PROGRAM P2_05_Process_Ctrl
VAR
	bWaitAferBatchClose			:BOOL;
	tonWaitAfterBatchClose		:TON;
END_VAR
VAR // added by the converter: edge detectors and wires of the graphical bodies
    _w1, _w2, _w3, _w4, _w5, _w6, _w7, _w8, _w9 : BOOL;
    _rt1, _rt2 : R_TRIG;
END_VAR

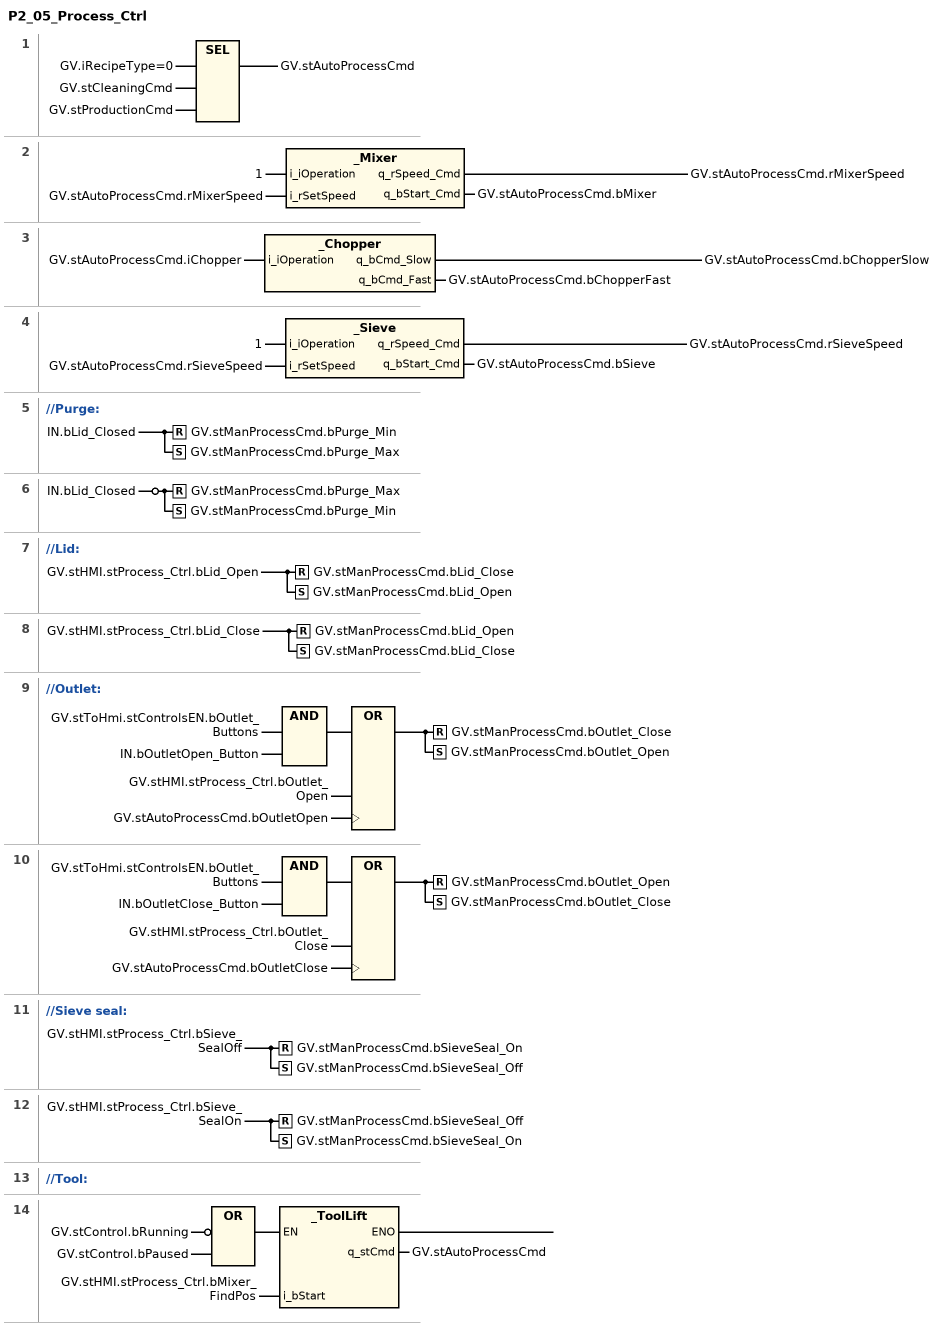
// NETWORK 1
GV.stAutoProcessCmd := SEL(GV.iRecipeType=0, GV.stCleaningCmd, GV.stProductionCmd);

// NETWORK 2
_Mixer(i_iOperation := 1, i_rSetSpeed := GV.stAutoProcessCmd.rMixerSpeed, q_bStart_Cmd => GV.stAutoProcessCmd.bMixer);
GV.stAutoProcessCmd.rMixerSpeed := _Mixer.q_rSpeed_Cmd;

// NETWORK 3
_Chopper(i_iOperation := GV.stAutoProcessCmd.iChopper, q_bCmd_Fast => GV.stAutoProcessCmd.bChopperFast);
GV.stAutoProcessCmd.bChopperSlow := _Chopper.q_bCmd_Slow;

// NETWORK 4
_Sieve(i_iOperation := 1, i_rSetSpeed := GV.stAutoProcessCmd.rSieveSpeed, q_bStart_Cmd => GV.stAutoProcessCmd.bSieve);
GV.stAutoProcessCmd.rSieveSpeed := _Sieve.q_rSpeed_Cmd;

// NETWORK 5
// label: //Purge
GV.stManProcessCmd.bPurge_Min R= IN.bLid_Closed;
GV.stManProcessCmd.bPurge_Max S= IN.bLid_Closed;

// NETWORK 6
_w1 := NOT IN.bLid_Closed;
GV.stManProcessCmd.bPurge_Max R= _w1;
GV.stManProcessCmd.bPurge_Min S= _w1;

// NETWORK 7
// label: //Lid
_w2 := GV.stHMI.stProcess_Ctrl.bLid_Open;
GV.stManProcessCmd.bLid_Close R= _w2;
GV.stManProcessCmd.bLid_Open S= _w2;

// NETWORK 8
_w3 := GV.stHMI.stProcess_Ctrl.bLid_Close;
GV.stManProcessCmd.bLid_Open R= _w3;
GV.stManProcessCmd.bLid_Close S= _w3;

// NETWORK 9
// label: //Outlet
_rt1(CLK := GV.stAutoProcessCmd.bOutletOpen);
_w4 := GV.stToHmi.stControlsEN.bOutlet_Buttons AND IN.bOutletOpen_Button OR GV.stHMI.stProcess_Ctrl.bOutlet_Open OR _rt1.Q;
GV.stManProcessCmd.bOutlet_Close R= _w4;
GV.stManProcessCmd.bOutlet_Open S= _w4;

// NETWORK 10
_rt2(CLK := GV.stAutoProcessCmd.bOutletClose);
_w5 := GV.stToHmi.stControlsEN.bOutlet_Buttons AND IN.bOutletClose_Button OR GV.stHMI.stProcess_Ctrl.bOutlet_Close OR _rt2.Q;
GV.stManProcessCmd.bOutlet_Open R= _w5;
GV.stManProcessCmd.bOutlet_Close S= _w5;

// NETWORK 11
// label: //Sieve seal
_w6 := GV.stHMI.stProcess_Ctrl.bSieve_SealOff;
GV.stManProcessCmd.bSieveSeal_On R= _w6;
GV.stManProcessCmd.bSieveSeal_Off S= _w6;

// NETWORK 12
_w7 := GV.stHMI.stProcess_Ctrl.bSieve_SealOn;
GV.stManProcessCmd.bSieveSeal_Off R= _w7;
GV.stManProcessCmd.bSieveSeal_On S= _w7;

// NETWORK 13
// label: //Tool

// NETWORK 14
IF NOT GV.stControl.bRunning OR GV.stControl.bPaused THEN
    _ToolLift(i_bStart := GV.stHMI.stProcess_Ctrl.bMixer_FindPos, q_stCmd => GV.stAutoProcessCmd);
END_IF

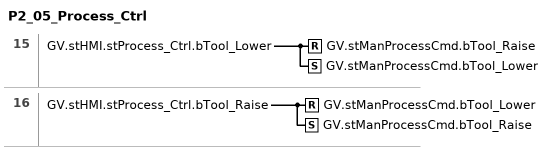
// NETWORK 15
_w8 := GV.stHMI.stProcess_Ctrl.bTool_Lower;
GV.stManProcessCmd.bTool_Raise R= _w8;
GV.stManProcessCmd.bTool_Lower S= _w8;

// NETWORK 16
_w9 := GV.stHMI.stProcess_Ctrl.bTool_Raise;
GV.stManProcessCmd.bTool_Lower R= _w9;
GV.stManProcessCmd.bTool_Raise S= _w9;

END_PROGRAM

(* stored: Version 1.1.0.1, ProductVersion 3.1.4026.13
   POU P2_05_Process_Ctrl: Id {e867a8fd-57c7-4ddf-9933-795cf451023c}, SpecialFunc None *)
